{attribute 'qualified_only'}
VAR_GLOBAL CONSTANT
	Itf0			: Result := -2; // Null Interface 
	Str0			: Result := -3; // Empty String
	ItfEq			: Result := -4; // Interfaces are equal
	NoMatch			: Result := -5; // No match
	Ptr0			: Result := -6; // Null Pointer
	InvRef			: Result := -7; // Invalid reference
	Ovf				: Result := -8; // Overflow/Out of bounds
	Udf				: Result := -9; // Undefined
	Idx				: Result := -10; // Index error
	TcLib			: Result := -11; // Error caused by TwinCAT libraries
	InfLoop			: Result := -12; // Potential infinity loop
	IncArg			: Result := -13; // Incorrect input argument
	Init			: Result := -14; // Initialisation error
	NotFound		: Result := -15; // Item not found
END_VAR

(* stored: Version 1.1.0.1
   GVL Err: Id {eeeb2f9f-a3e9-42a4-bf82-bcee2d1ba591} *)
